// Mitsubishi GX Works2 project: gruop11   PLC: FX3G

// global labels: Global1
VAR_GLOBAL
  Start_Workday AT X007 : BOOL;
  Chocolate_input AT D1100 : REAL;
  Chocolate_container AT D5000 : REAL;
  Nuts_input AT D1110 : REAL;
  Nuts_container AT D5010 : REAL;
  Pistachios_input AT D1120 : REAL;
  Pistachios_container AT D5020 : REAL;
  Kadaif_input AT D1130 : REAL;
  Kadaif_container AT D5030 : REAL;
  Working_day_light AT Y007 : BOOL;
  End_day AT M7 : BOOL;
  Emergency_switch AT X005 : BOOL;
  Out_of_stock AT M5 : BOOL;
  Melting AT X001 : BOOL;
  Melting_container AT D5040 : REAL;
  Start_melting AT X001 : BOOL;
  Melting_light AT Y001 : BOOL;
  Temp_sensor AT X002 : BOOL;
  Melting_light_P AT M1 : BOOL;
  LLLL AT Y003 : BOOL;
  Temp_to_casting AT M2 : BOOL;
  Table_pos AT X003 : BOOL;
  Const_Const AT E400.0 : REAL;
  Meltimg_cont AT D5040 : REAL;
  Tser AT Y011 : BOOL;
  Meltimg_containe : REAL;
  Start_casting AT M2 : BOOL;
  Table_1 AT D5060 : REAL;
  Const_add_table AT E100.0 : REAL;
  Table_3 AT D5080 : REAL;
  Table_2 AT D5070 : REAL;
  Table_4 AT D5090 : REAL;
  TS_40 AT TS40 : BOOL;
  Casting_light AT Y002 : BOOL;
  Const_time AT E40 : REAL;
  TC_1 AT TC1 : BOOL;
END_VAR
VAR_GLOBAL CONSTANT
  Const_40_casting : REAL := 40.0;
END_VAR
VAR_GLOBAL
  TS_1 AT TS1 : BOOL;
  Analog_1 AT X004 : BOOL;
END_VAR
VAR_GLOBAL CONSTANT
  Const_5 : REAL := 5.1;
END_VAR
VAR_GLOBAL
  Choose_dxb AT M4 : BOOL;
  Choose_nuts AT M6 : BOOL;
  Test AT Y011 : BOOL;
  test1 AT Y010 : BOOL;
  Norm_input AT D1510 : REAL;
  Save_analog AT D1500 : REAL;
  Nuts_cream AT D6010 : REAL;
END_VAR
VAR_GLOBAL CONSTANT
  Add_nuts : REAL := 20;
  Add_pis : REAL := 100;
  Nuts_sub : REAL := 100;
  Pistachios_sub : REAL := 100;
END_VAR
VAR_GLOBAL
  dxb_cream AT D6000 : REAL;
END_VAR
VAR_GLOBAL CONSTANT
  Add_nuts_dxb : REAL := 20;
  Add_nuts_nuts : REAL := 100;
  Add_pis_dxb : REAL := 120;
  Add_kadaif_dxb : REAL := 60;
  Nuts_dxb_sub : REAL := 20;
  Pistachios_dxb_sub : REAL := 120;
  kadaif_dxb_sub : REAL := 60;
END_VAR
VAR_GLOBAL
  tast AT Y010 : BOOL;
  ttttt AT Y011 : BOOL;
  TC_5 AT TC5 : BOOL;
  blink_timer AT TS5 : BOOL;
  start_blink AT M10 : BOOL;
  TC_3 AT TC3 : BOOL;
  Y3_timer AT TS3 : BOOL;
  light_3 AT Y003 : BOOL;
  TC_4 AT TC4 : BOOL;
  Y4_timer AT TS4 : BOOL;
  light_4 AT Y004 : BOOL;
  Colling AT X006 : BOOL;
  Start_Colling AT X006 : BOOL;
  TC_6 AT TC6 : BOOL;
  Cooling_light AT Y006 : BOOL;
  Start_Coolling AT X006 : BOOL;
  Finsh_cream AT M11 : BOOL;
  Y6_timer AT TS6 : BOOL;
END_VAR
VAR_GLOBAL CONSTANT
  Timer_3sec : INT := 30;
  Timer_blink5 : INT := 5;
  Timer_5sec : INT := 50;
END_VAR
VAR_GLOBAL
  Finsh_Cooling AT M12 : BOOL;
  pack_package AT CC1 : BOOL;
  count_table AT X000 : BOOL;
  pack_single_table AT CC0 : BOOL;
END_VAR
VAR_GLOBAL CONSTANT
  package_4 : INT := 4;
  cont_table : INT := 1;
  add_table : INT := 1;
END_VAR
VAR_GLOBAL
  pack_package_cs AT CS1 : BOOL;
END_VAR
VAR_GLOBAL CONSTANT
  add_packge : INT := 4;
END_VAR
VAR_GLOBAL
  package_container AT D7000 : REAL;
END_VAR
VAR_GLOBAL CONSTANT
  Const_package : REAL := 1;
END_VAR
VAR_GLOBAL
  pack_single_table_cs AT CS0 : BOOL;
  packing_light AT Y005 : BOOL;
END_VAR
VAR_GLOBAL CONSTANT
  Const_40 : INT := 40;
END_VAR
VAR_GLOBAL
  Analog_2 AT D8282 : INT;
  Total_package AT D7020 : REAL;
  show_answer AT D7010 : REAL;
END_VAR
VAR_GLOBAL CONSTANT
  Const_40_normal : REAL := 40.0;
END_VAR
VAR_GLOBAL
  Count_rest AT M13 : BOOL;
  Const_100 AT E100 : REAL;
  Const_120 AT E120 : REAL;
END_VAR
VAR_GLOBAL CONSTANT
  Const_399 : REAL := 399;
  Const_99 : REAL := 99;
  Const_119 : REAL := 119;
END_VAR
VAR_GLOBAL
  Analog_input1 AT D8280 : INT;
END_VAR

// task Task_01 (event TRUE, interval 0, priority 31): POU_01

PROGRAM POU_01
VAR
  Meltimg_container : REAL;
END_VAR
VAR CONSTANT
  Const_400 : WORD := 40;
END_VAR
VAR
  time40 : TIME;
  TC_40 : TIME;
END_VAR
VAR CONSTANT
  Const_60 : REAL := 60;
  Const_59 : REAL := 59;
END_VAR
(* structured ladder/FBD written out as ST: instructions are called as NAME(EN, inputs, outputs); _pN, _eN, _tN stand for wires *)
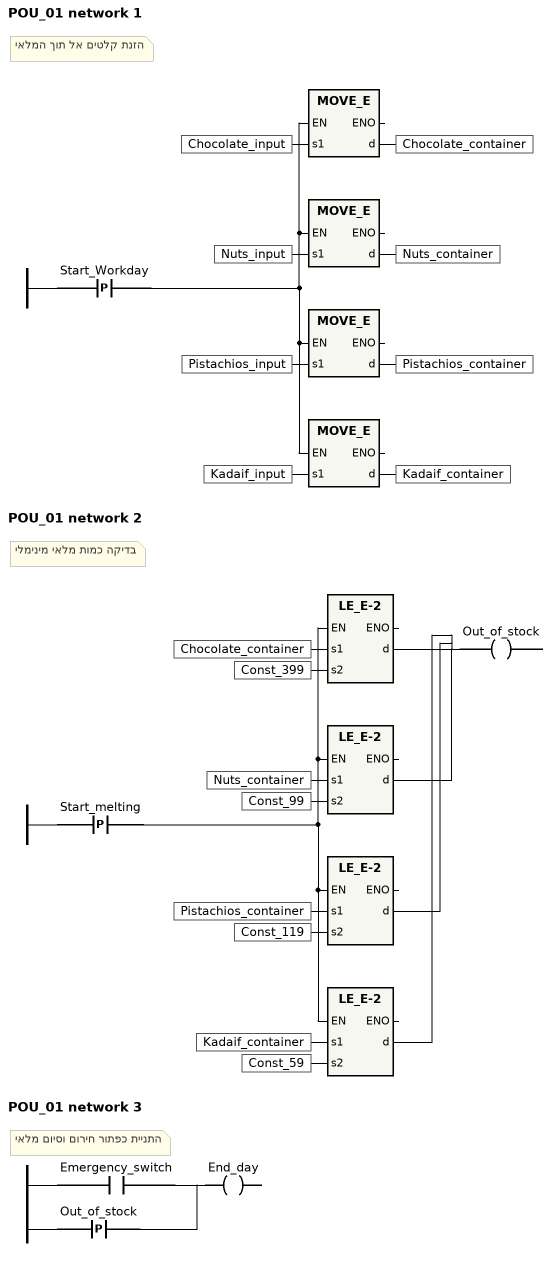
(* network 1 *)
(* הזנת קלטים אל תוך המלאי *)
_p1 := LDP(TRUE, Start_Workday);
MOVE_E(_p1, Chocolate_input, Chocolate_container);
MOVE_E(_p1, Nuts_input, Nuts_container);
MOVE_E(_p1, Pistachios_input, Pistachios_container);
MOVE_E(_p1, Kadaif_input, Kadaif_container);
(* network 2 *)
(* בדיקה כמות מלאי מינימלי *)
_p1 := LDP(TRUE, Start_melting);
LE_E(_p1, Chocolate_container, Const_399, _t2);
LE_E(_p1, Nuts_container, Const_99, _t3);
LE_E(_p1, Pistachios_container, Const_119, _t4);
LE_E(_p1, Kadaif_container, Const_59, _t5);
Out_of_stock := _t2 OR _t3 OR _t4 OR _t5;
(* network 3 *)
(* התניית כפתור חירום וסיום מלאי *)
End_day := Emergency_switch OR LDP(TRUE, Out_of_stock);
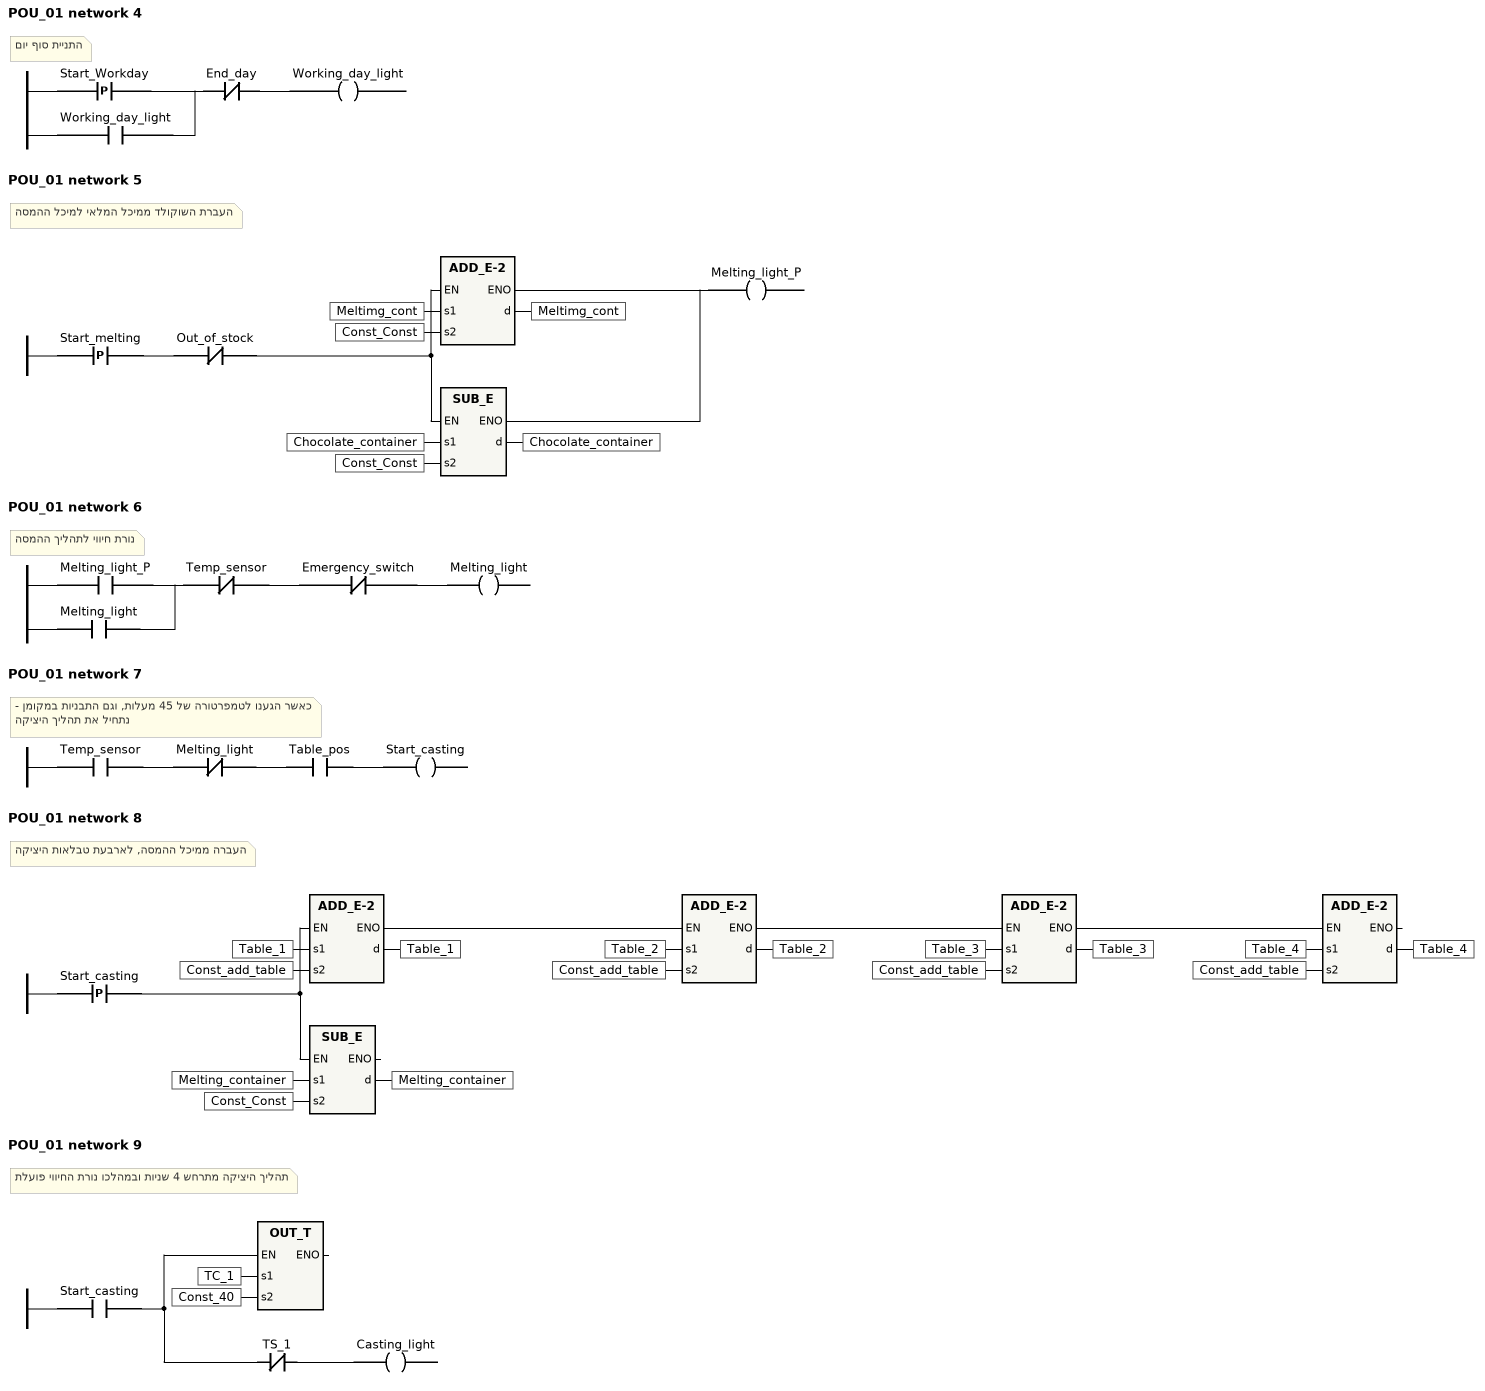
(* network 4 *)
(* התניית סוף יום *)
Working_day_light := (LDP(TRUE, Start_Workday) OR Working_day_light) AND NOT End_day;
(* network 5 *)
(* העברת השוקולד ממיכל המלאי למיכל ההמסה *)
_p1 := LDP(TRUE, Start_melting) AND NOT Out_of_stock;
_e2 := ADD_E(_p1, Meltimg_cont, Const_Const, Meltimg_cont);
_e3 := SUB_E(_p1, Chocolate_container, Const_Const, Chocolate_container);
Melting_light_P := _e2 OR _e3;
(* network 6 *)
(* נורת חיווי לתהליך ההמסה *)
Melting_light := ((Melting_light_P OR Melting_light) AND NOT Temp_sensor) AND NOT Emergency_switch;
(* network 7 *)
(* כאשר הגענו לטמפרטורה של 45 מעלות, וגם התבניות במקומן - נתחיל את תהליך היציקה *)
Start_casting := Temp_sensor AND NOT Melting_light AND Table_pos;
(* network 8 *)
(* העברה ממיכל ההמסה, לארבעת טבלאות היציקה *)
_p1 := LDP(TRUE, Start_casting);
_e2 := ADD_E(_p1, Table_1, Const_add_table, Table_1);
_e3 := ADD_E(_e2, Table_2, Const_add_table, Table_2);
_e4 := ADD_E(_e3, Table_3, Const_add_table, Table_3);
ADD_E(_e4, Table_4, Const_add_table, Table_4);
SUB_E(_p1, Melting_container, Const_Const, Melting_container);
(* network 9 *)
(* תהליך היציקה מתרחש 4 שניות ובמהלכו נורת החיווי פועלת *)
OUT_T(Start_casting, TC_1, Const_40);
Casting_light := Start_casting AND NOT TS_1;
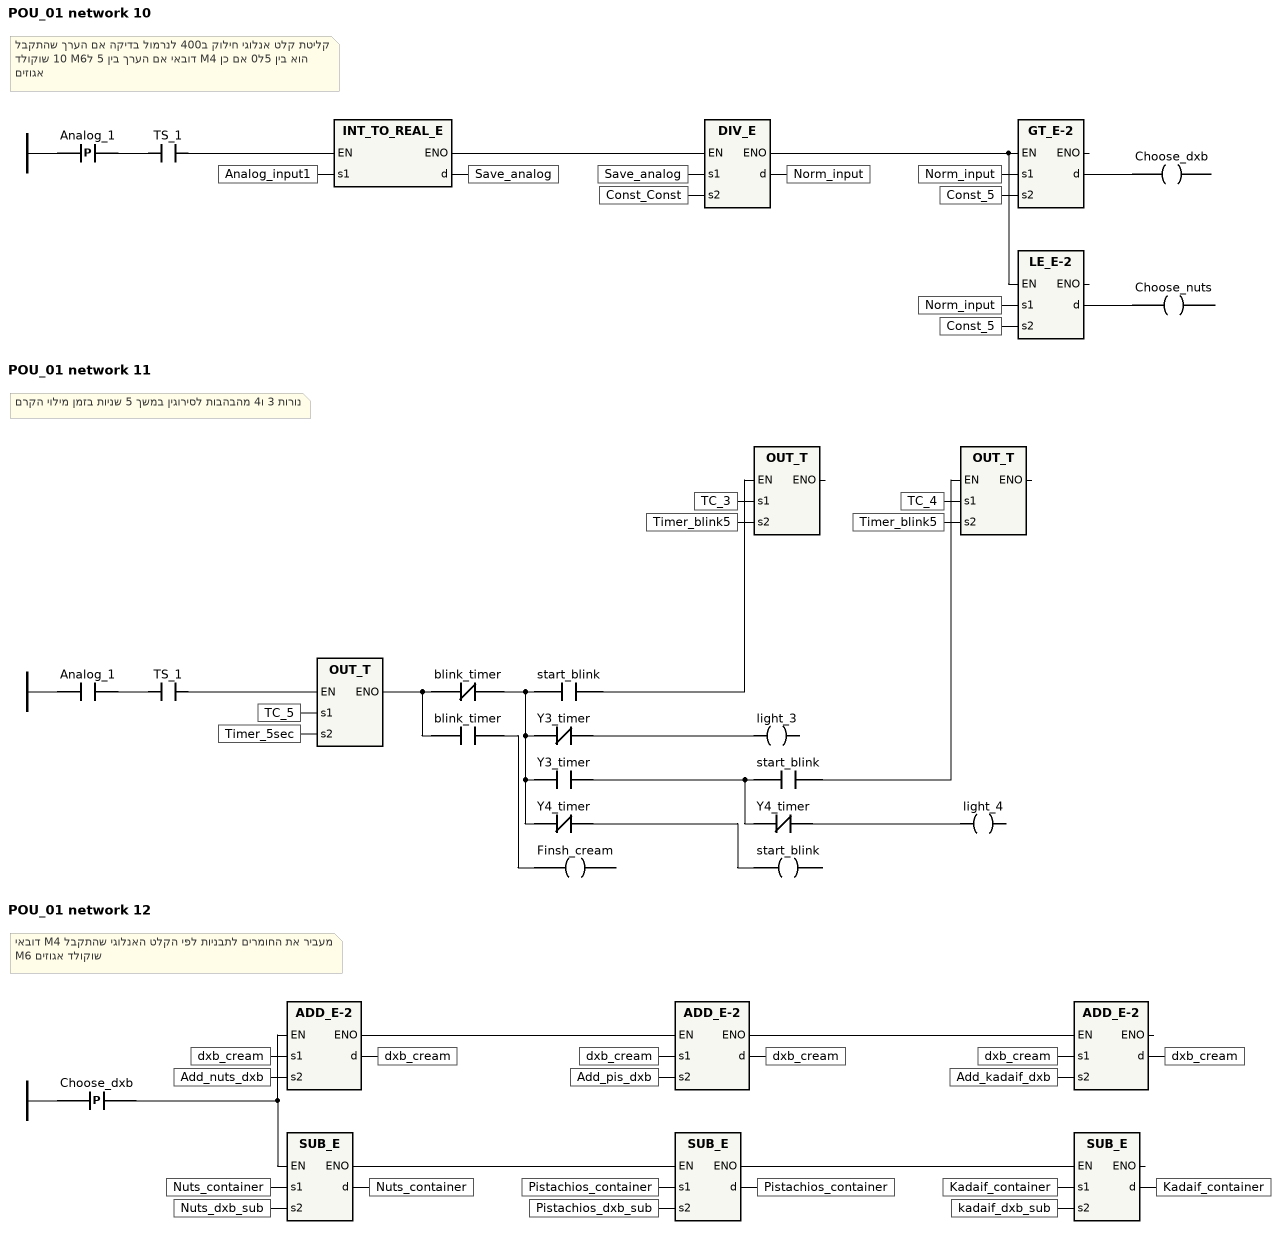
(* network 10 *)
(* קליטת קלט אנלוגי חילוק ב400 לנרמול בדיקה אם הערך שהתקבל הוא בין 5ל0 אם כן M4 דובאי אם הערך בין 5 ל10 M6 שוקולד אגוזים *)
_e1 := INT_TO_REAL_E(LDP(TRUE, Analog_1) AND TS_1, Analog_input1, Save_analog);
_e2 := DIV_E(_e1, Save_analog, Const_Const, Norm_input);
GT_E(_e2, Norm_input, Const_5, _t3);
Choose_dxb := _t3;
LE_E(_e2, Norm_input, Const_5, _t4);
Choose_nuts := _t4;
(* network 11 *)
(* נורות 3 ו4 מהבהבות לסירוגין במשך 5 שניות בזמן מילוי הקרם *)
_e1 := OUT_T(Analog_1 AND TS_1, TC_5, Timer_5sec);
_p2 := _e1 AND NOT blink_timer;
OUT_T(_p2 AND start_blink, TC_3, Timer_blink5);
light_3 := _p2 AND NOT Y3_timer;
_p3 := _p2 AND Y3_timer;
OUT_T(_p3 AND start_blink, TC_4, Timer_blink5);
light_4 := _p3 AND NOT Y4_timer;
start_blink := _p2 AND NOT Y4_timer;
Finsh_cream := _e1 AND blink_timer;
(* network 12 *)
(* מעביר את החומרים לתבניות לפי הקלט האנלוגי שהתקבל M4 דובאי             M6 שוקולד אגוזים *)
_p1 := LDP(TRUE, Choose_dxb);
_e2 := ADD_E(_p1, dxb_cream, Add_nuts_dxb, dxb_cream);
_e3 := ADD_E(_e2, dxb_cream, Add_pis_dxb, dxb_cream);
ADD_E(_e3, dxb_cream, Add_kadaif_dxb, dxb_cream);
_e4 := SUB_E(_p1, Nuts_container, Nuts_dxb_sub, Nuts_container);
_e5 := SUB_E(_e4, Pistachios_container, Pistachios_dxb_sub, Pistachios_container);
SUB_E(_e5, Kadaif_container, kadaif_dxb_sub, Kadaif_container);
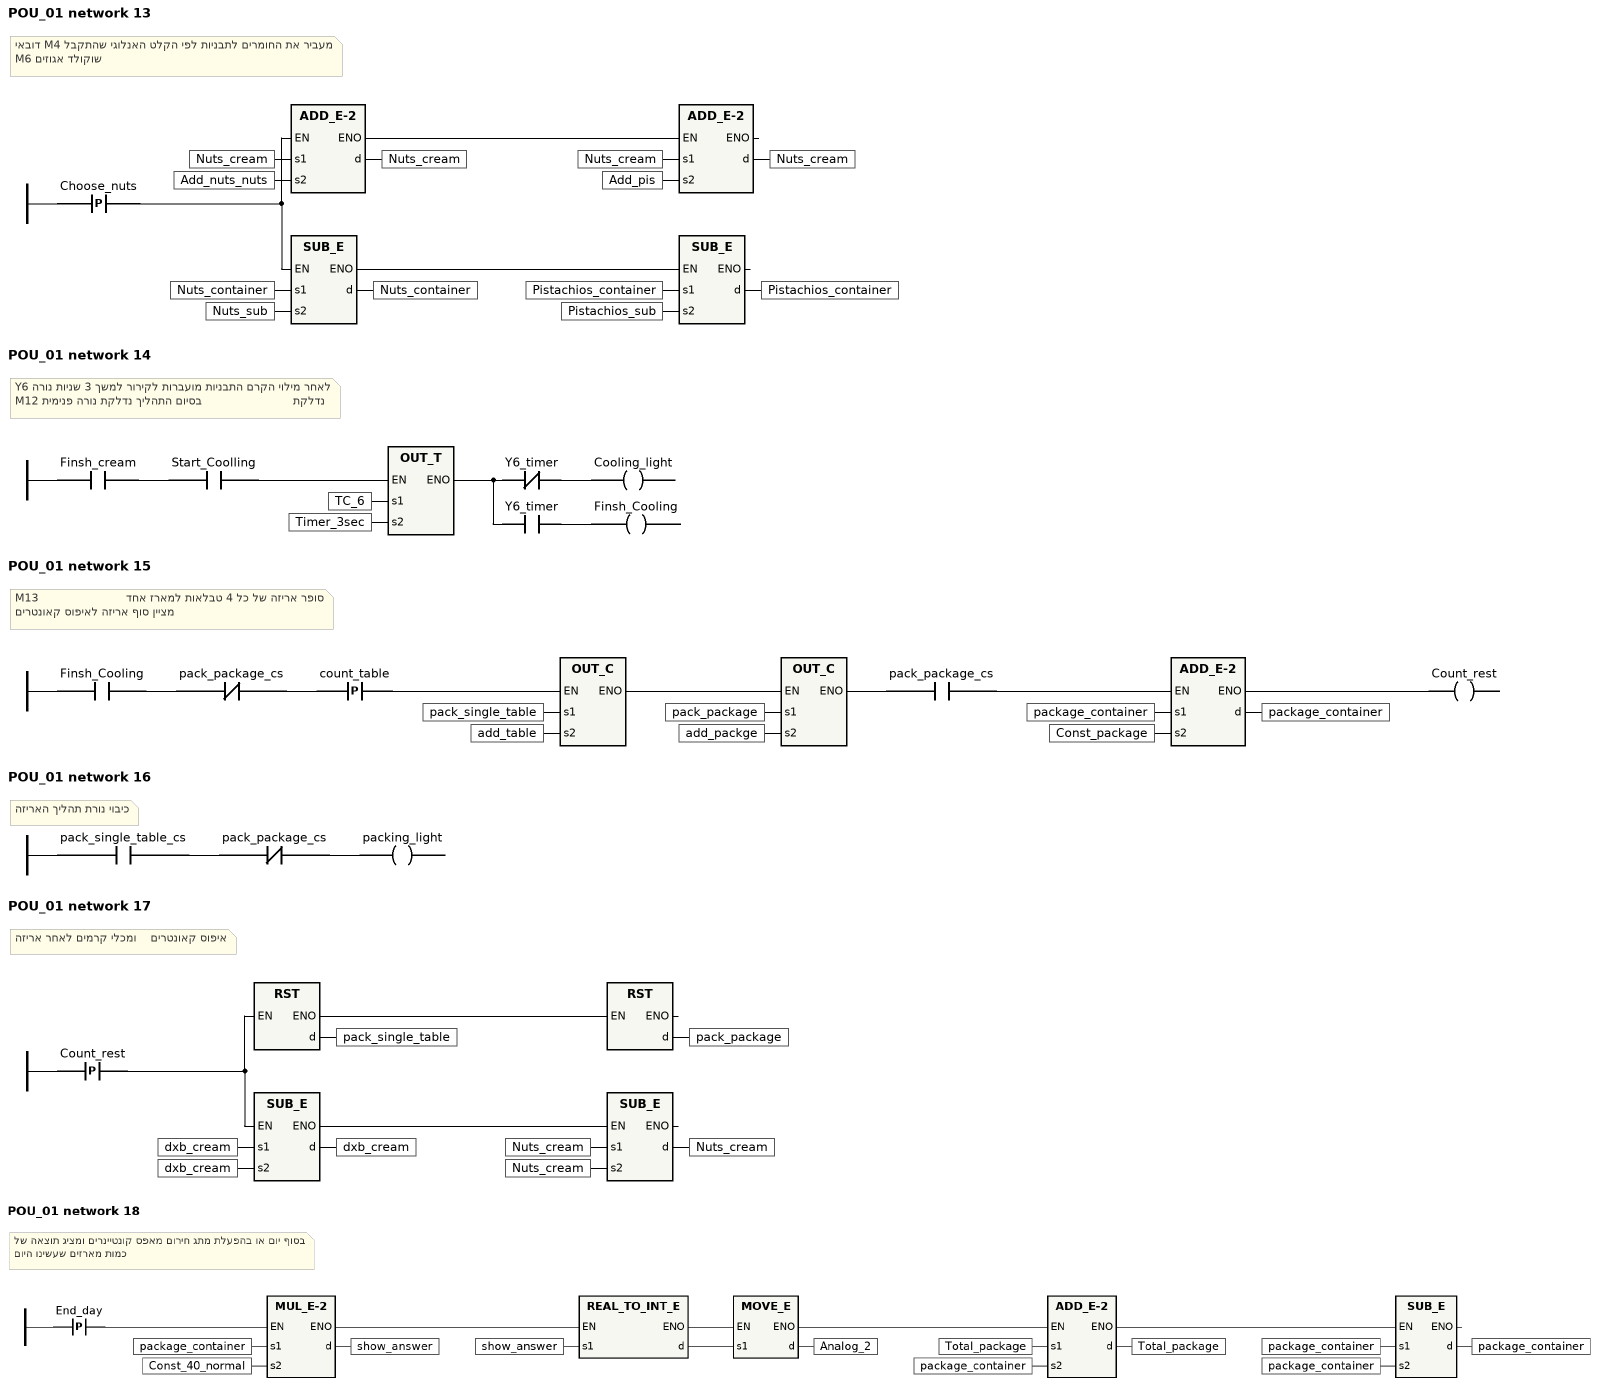
(* network 13 *)
(* מעביר את החומרים לתבניות לפי הקלט האנלוגי שהתקבל M4 דובאי             M6 שוקולד אגוזים *)
_p1 := LDP(TRUE, Choose_nuts);
_e2 := ADD_E(_p1, Nuts_cream, Add_nuts_nuts, Nuts_cream);
ADD_E(_e2, Nuts_cream, Add_pis, Nuts_cream);
_e3 := SUB_E(_p1, Nuts_container, Nuts_sub, Nuts_container);
SUB_E(_e3, Pistachios_container, Pistachios_sub, Pistachios_container);
(* network 14 *)
(* לאחר מילוי הקרם התבניות מועברות לקירור למשך 3 שניות נורה Y6 נדלקת                          בסיום התהליך נדלקת נורה פנימית M12 *)
_e1 := OUT_T(Finsh_cream AND Start_Coolling, TC_6, Timer_3sec);
Cooling_light := _e1 AND NOT Y6_timer;
Finsh_Cooling := _e1 AND Y6_timer;
(* network 15 *)
(* סופר אריזה של כל 4 טבלאות למארז אחד                         M13 מציין סוף אריזה לאיפוס קאונטרים *)
_e1 := OUT_C(Finsh_Cooling AND NOT pack_package_cs AND LDP(TRUE, count_table), pack_single_table, add_table);
_e2 := OUT_C(_e1, pack_package, add_packge);
_e3 := ADD_E(_e2 AND pack_package_cs, package_container, Const_package, package_container);
Count_rest := _e3;
(* network 16 *)
(* כיבוי נורת תהליך האריזה *)
packing_light := pack_single_table_cs AND NOT pack_package_cs;
(* network 17 *)
(* איפוס קאונטרים    ומכלי קרמים לאחר אריזה *)
_p1 := LDP(TRUE, Count_rest);
_e2 := RST(_p1, pack_single_table);
RST(_e2, pack_package);
_e3 := SUB_E(_p1, dxb_cream, dxb_cream, dxb_cream);
SUB_E(_e3, Nuts_cream, Nuts_cream, Nuts_cream);
(* network 18 *)
(* בסוף יום או בהפעלת מתג חירום מאפס קונטיינרים ומציג תוצאה של כמות מארזים שעשינו היום *)
_e1 := MUL_E(LDP(TRUE, End_day), package_container, Const_40_normal, show_answer);
_e3 := REAL_TO_INT_E(_e1, show_answer, _t2);
_e4 := MOVE_E(_e3, _t2, Analog_2);
_e5 := ADD_E(_e4, Total_package, package_container, Total_package);
SUB_E(_e5, package_container, package_container, package_container);
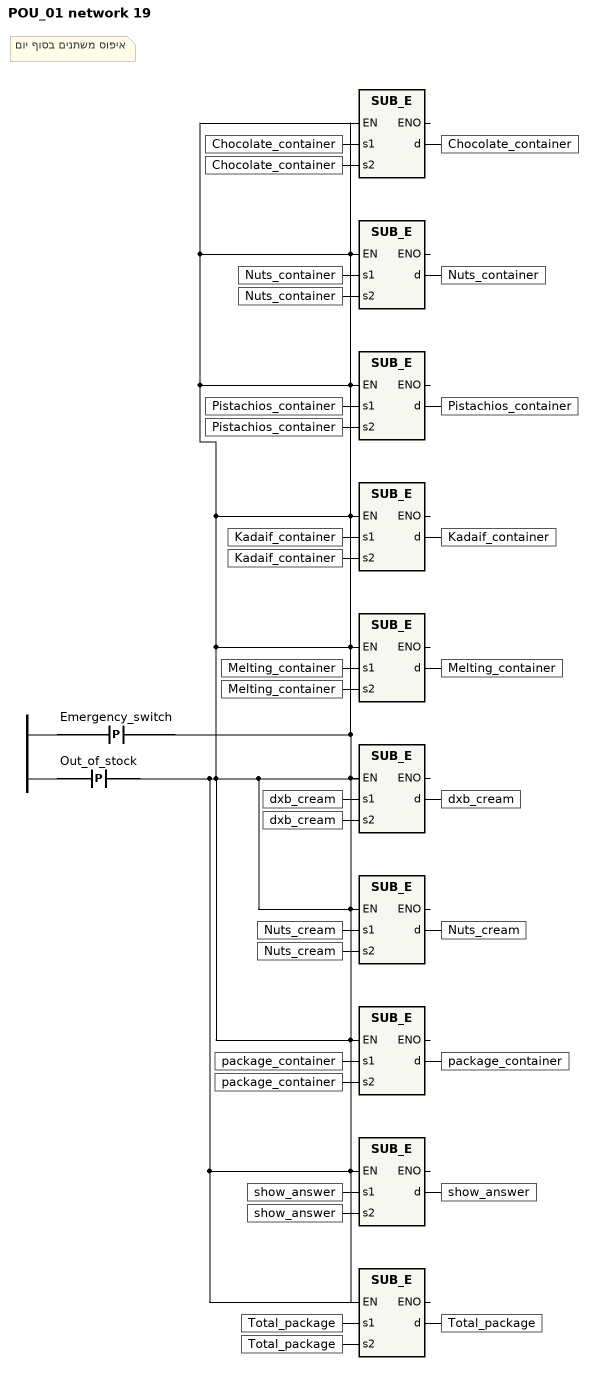
(* network 19 *)
(* איפוס משתנים בסוף יום *)
_p1 := LDP(TRUE, Emergency_switch) OR LDP(TRUE, Out_of_stock);
SUB_E(_p1, Chocolate_container, Chocolate_container, Chocolate_container);
SUB_E(_p1, Nuts_container, Nuts_container, Nuts_container);
SUB_E(_p1, Pistachios_container, Pistachios_container, Pistachios_container);
SUB_E(_p1, Kadaif_container, Kadaif_container, Kadaif_container);
SUB_E(_p1, Melting_container, Melting_container, Melting_container);
SUB_E(_p1, dxb_cream, dxb_cream, dxb_cream);
SUB_E(_p1, Nuts_cream, Nuts_cream, Nuts_cream);
SUB_E(_p1, package_container, package_container, package_container);
SUB_E(_p1, show_answer, show_answer, show_answer);
SUB_E(_p1, Total_package, Total_package, Total_package);
END_PROGRAM
